TYPE ZCom :
STRUCT
  // module context
  App : ZApplication.ApplicationComPublish;
  Alarming : ZApplication.AlarmingCom;
  Messages : ZApplication.MessagingCom;
  
  // unit context
  Unit : ZComUnit;

END_STRUCT
END_TYPE

(* stored: Version 1.1.0.1
   DUT ZCom: Id {d04e1d47-2a69-4b4e-9861-8b7cce8940f1} *)
